FUNCTION TestFunc (* Function with empty body *)
  (* Standard: 61499-1 *)
  (* Version 1.0, 2026-07-06, Franz Höpfinger, Meisterschulen am Ostbahnhof *)
  PACKAGE Meins;
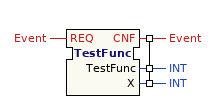
  EVENT_INPUT
    REQ;
  END_EVENT
  EVENT_OUTPUT
    CNF WITH TestFunc, X;
  END_EVENT
  VAR_OUTPUT
    TestFunc : INT;
    X : INT := 5;
  END_VAR
  BODY IN ST:
PACKAGE Meins;

(*
 * Function with empty body
 *)
FUNCTION TestFunc : INT

VAR_OUTPUT
	X : INT := 5;
END_VAR

TestFunc := 5;
X := 7;
END_FUNCTION
  END_BODY
END_FUNCTION
